(* CoDeSys 2.3.9.37 project: Cap8_7.pro *)
(* Libraries: Standard.lib 4.10.05 12:14:46 *)

(* Global variable list: Global_Variables *)
VAR_GLOBAL
      (* Entradas *)
	A1: BOOL;
	B1: BOOL;
	A2: BOOL;
	B2: BOOL;

      (* Salidas *)
	LuzVerde: BOOL;
	LuzAmarilla: BOOL;
	LuzRoja: BOOL;
       AvisoLleno:BOOL;

    (* Otras variables *)
       Aforo: INT;   (* Aforo máximo. Hay que darle valor *)
	Contador: CTUD;  (*Contador de  personas dentro *)
       Visitas:CTU;  (* Contados de número total de visitas *)
        Temporizador:TON; (*Temporizador de museo lleno *)

END_VAR

(* POU PLC_PRG, IL *)
PROGRAM PLC_PRG
VAR
END_VAR
	CAL		Animacion
END_PROGRAM

(* POU Animacion, ST *)
PROGRAM Animacion
VAR
      velocidad:INT:=2;

  (* Variables para puerta izquierda *)
   persona1xIzq:INT:=-1000;
   persona1yIzq:INT:=0;
  persona2xIzq:INT:=-1000;
   persona2yIzq:INT:=0;
	Ocupado1: BOOL;
       EntraPersona1:BOOL;
	EntrandoPersona1: BOOL;
	SalePersona1: BOOL;
	SaliendoPersona1: BOOL;
       EntraSale1:BOOL;
       EntrandoSaliendo1:BOOL;
	SaleEntra1: BOOL;
	SaliendoEntrando1: BOOL;

  (* Variables para puerta derecha *)
   persona1xDer:INT:=-1000;
   persona1yDer:INT:=0;
  persona2xDer:INT:=-1000;
   persona2yDer:INT:=0;
	Ocupado2: BOOL;
       EntraPersona2:BOOL;
	EntrandoPersona2: BOOL;
	SalePersona2: BOOL;
	SaliendoPersona2: BOOL;
       EntraSale2:BOOL;
       EntrandoSaliendo2:BOOL;
	SaleEntra2: BOOL;
	SaliendoEntrando2: BOOL;

END_VAR
(* Entrada puerta izquierda *)
IF Ocupado1=FALSE THEN

   IF EntraPersona1 AND LuzRoja=FALSE THEN
       EntrandoPersona1:=TRUE;
       persona1xIzq:=0;
       Ocupado1:=TRUE;
   END_IF

  IF SalePersona1 (* AND Contador.CV>0*) THEN
     SaliendoPersona1:=TRUE;
      persona2xIzq:=0;
      Ocupado1:=TRUE;
   END_IF

  IF EntraSale1 AND LuzRoja=FALSE (*AND Contador.CV>0*) THEN
   EntrandoSaliendo1:=TRUE;
   persona1xIzq:=30;
   persona2xIzq:=0;
   Ocupado1:=TRUE;
  END_IF

  IF SaleEntra1 AND LuzRoja=FALSE (*AND Contador.CV>0*) THEN
   SaliendoEntrando1:=TRUE;
   persona1xIzq:=0;
   persona2xIzq:=-10;
   Ocupado1:=TRUE;
  END_IF

END_IF



IF EntrandoPersona1 THEN
    persona1xIzq:=persona1xIzq+velocidad;
    IF persona1xIzq>70 AND persona1xIzq<97 THEN
      A1:=TRUE;
    ELSE
       A1:=FALSE;
    END_IF
    IF persona1xIzq>=75 AND persona1xIzq<105 THEN
      B1:=TRUE;
    ELSE
       B1:=FALSE;
    END_IF
   IF persona1xIzq>150 THEN
      EntrandoPersona1:=FALSE;
      persona1xIzq:=-1000;
      Ocupado1:=FALSE;
   END_IF
 END_IF


IF SaliendoPersona1 THEN
    persona2xIzq:=persona2xIzq-velocidad;
    IF persona2xIzq<-60 AND persona2xIzq>-87 THEN
      B1:=TRUE;
    ELSE
       B1:=FALSE;
    END_IF
    IF persona2xIzq<=-65 AND persona2xIzq>-95 THEN
      A1:=TRUE;
    ELSE
       A1:=FALSE;
    END_IF
   IF persona2xIzq<-150 THEN
      SaliendoPersona1:=FALSE;
      persona2xIzq:=-1000;
      Ocupado1:=FALSE;
   END_IF
 END_IF


IF EntrandoSaliendo1 OR SaliendoEntrando1 THEN

    persona2xIzq:=persona2xIzq-velocidad;
    persona1xIzq:=persona1xIzq+velocidad;
    IF (persona2xIzq<-60 AND persona2xIzq>-87) OR (  persona1xIzq>=75 AND persona1xIzq<105) THEN
      B1:=TRUE;
    ELSE
       B1:=FALSE;
    END_IF
    IF(persona2xIzq<=-65 AND persona2xIzq>-95) OR ( persona1xIzq>70 AND persona1xIzq<97) THEN
      A1:=TRUE;
    ELSE
       A1:=FALSE;
    END_IF

   IF (persona2xIzq<-150) AND (persona1xIzq>150)  THEN
      EntrandoSaliendo1:=FALSE;
     SaliendoEntrando1:=FALSE;
       persona1xIzq:=-1000;
      persona2xIzq:=-1000;
      Ocupado1:=FALSE;
   END_IF
 END_IF





(* Entrada puerta derecha *)
IF Ocupado2=FALSE THEN

   IF EntraPersona2 AND LuzRoja=FALSE THEN
       EntrandoPersona2:=TRUE;
       persona1xDer:=0;
       Ocupado2:=TRUE;
   END_IF

  IF SalePersona2 (*AND Contador.CV>0*) THEN
     SaliendoPersona2:=TRUE;
      persona2xDer:=0;
      Ocupado2:=TRUE;
   END_IF

  IF EntraSale2 AND LuzRoja=FALSE (*AND Contador.CV>0*) THEN
   EntrandoSaliendo2:=TRUE;
   persona1xDer:=30;
   persona2xDer:=0;
   Ocupado2:=TRUE;
  END_IF

  IF SaleEntra2 AND LuzRoja=FALSE (* AND Contador.CV>0 *) THEN
   SaliendoEntrando2:=TRUE;
   persona1xDer:=0;
   persona2xDer:=-10;
   Ocupado2:=TRUE;
  END_IF

END_IF



IF EntrandoPersona2 THEN
    persona1xDer:=persona1xDer+velocidad;
    IF persona1xDer>70 AND persona1xDer<97 THEN
      A2:=TRUE;
    ELSE
       A2:=FALSE;
    END_IF
    IF persona1xDer>=75 AND persona1xDer<105 THEN
      B2:=TRUE;
    ELSE
       B2:=FALSE;
    END_IF
   IF persona1xDer>150 THEN
      EntrandoPersona2:=FALSE;
      persona1xDer:=-1000;
      Ocupado2:=FALSE;
   END_IF
 END_IF


IF SaliendoPersona2 THEN
    persona2xDer:=persona2xDer-velocidad;
    IF persona2xDer<-60 AND persona2xDer>-87 THEN
      B2:=TRUE;
    ELSE
       B2:=FALSE;
    END_IF
    IF persona2xDer<=-65 AND persona2xDer>-95 THEN
      A2:=TRUE;
    ELSE
       A2:=FALSE;
    END_IF
   IF persona2xDer<-150 THEN
      SaliendoPersona2:=FALSE;
      persona2xDer:=-1000;
      Ocupado2:=FALSE;
   END_IF
 END_IF


IF EntrandoSaliendo2 OR SaliendoEntrando2 THEN

    persona2xDer:=persona2xDer-velocidad;
    persona1xDer:=persona1xDer+velocidad;
    IF (persona2xDer<-60 AND persona2xDer>-87) OR (  persona1xDer>=75 AND persona1xDer<105) THEN
      B2:=TRUE;
    ELSE
       B2:=FALSE;
    END_IF
    IF(persona2xDer<=-65 AND persona2xDer>-95) OR ( persona1xDer>70 AND persona1xDer<97) THEN
      A2:=TRUE;
    ELSE
       A2:=FALSE;
    END_IF

   IF (persona2xDer<-150) AND (persona1xDer>150)  THEN
      EntrandoSaliendo2:=FALSE;
     SaliendoEntrando2:=FALSE;
       persona1xDer:=-1000;
      persona2xDer:=-1000;
      Ocupado2:=FALSE;
   END_IF
 END_IF
END_PROGRAM

(* Visualisation Museo
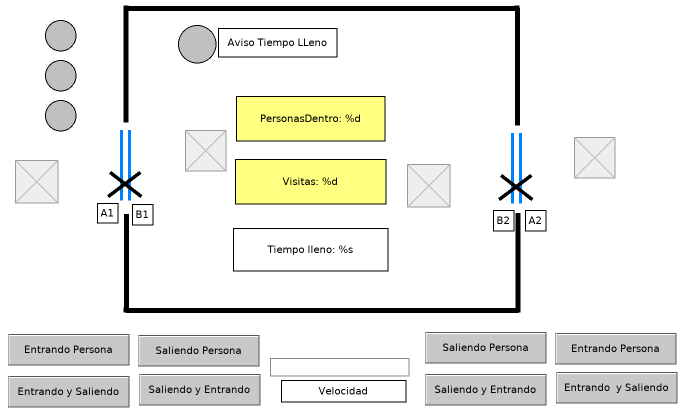
ellipse at (50,40)-(81,71): alarm colour if LuzRoja
ellipse at (50,80)-(81,111): alarm colour if LuzAmarilla
ellipse at (50,120)-(81,151): alarm colour if LuzVerde
rectangle at (241,116)-(390,161): text "PersonasDentro: %d"; shows contador.CV
bitmap at (20,180)-(61,221): SILHOUETTE_MAN_WALKING_BACKPACK.TIF
polyline at (126,150)-(126,220): alarm colour if A1
polyline at (134,150)-(134,220): alarm colour if B1
rectangle at (102,223)-(123,243): text "A1"
rectangle at (137,224)-(158,245): text "B1"
button at (13,354)-(134,385): text "Entrando Persona"; taps Animacion.EntraPersona1
bitmap at (190,150)-(231,191): DibujosEj6\persona2.bmp
button at (143,355)-(264,386): text "Saliendo Persona"; taps Animacion.SalePersona1
button at (13,396)-(134,427): text "Entrando y Saliendo"; taps Animacion.EntraSale1
button at (144,394)-(265,425): text "Saliendo y Entrando"; taps Animacion.SaleEntra1
rectangle at (286,400)-(411,422): text "Velocidad"
polyline at (115,192)-(146,216): alarm colour if LuzRoja
polyline at (113,192)-(145,216): alarm colour if luzroja
rectangle at (240,179)-(391,224): text "Visitas: %d"; shows visitas.CV
bitmap at (20,180)-(63,223): DibujosEj6\persona1.bmp
ellipse at (183,45)-(221,83): alarm colour if AvisoLleno
rectangle at (223,48)-(342,77): text "Aviso Tiempo LLeno"
rectangle at (238,248)-(393,291): text "Tiempo lleno: %s"; shows Temporizador.ET
polyline at (517,153)-(517,223): alarm colour if A2
polyline at (525,153)-(525,223): alarm colour if B2
rectangle at (498,230)-(519,251): text "B2"
polyline at (506,195)-(537,219): alarm colour if LuzRoja
polyline at (504,195)-(536,219): alarm colour if luzroja
rectangle at (530,230)-(551,251): text "A2"
button at (430,352)-(551,383): text "Saliendo Persona"; taps Animacion.EntraPersona2
button at (560,353)-(681,384): text "Entrando Persona"; taps Animacion.SalePersona2
button at (430,394)-(551,425): text "Saliendo y Entrando"; taps Animacion.EntraSale2
button at (561,392)-(682,423): text "Entrando  y Saliendo"; taps Animacion.SaleEntra2
bitmap at (412,184)-(455,227): DibujosEj6\persona1.bmp
bitmap at (579,157)-(620,198): DibujosEj6\persona2.bmp
3 more shapes without text or variables
*)
